(* IEC 61131-3 sources: OLIA-RU/Lirics/OpenPLC_Runtime/Projects/ModbusTCP_slave_test/build, 2 files *)

(* ---- plc.st ---- *)
TYPE
  LOGLEVEL : (CRITICAL, WARNING, INFO, DEBUG) := INFO;
END_TYPE

FUNCTION_BLOCK LOGGER
  VAR_INPUT
    TRIG : BOOL;
    MSG : STRING;
    LEVEL : LOGLEVEL := INFO;
  END_VAR
  VAR
    TRIG0 : BOOL;
  END_VAR

  IF TRIG AND NOT TRIG0 THEN
  {{
   LogMessage(GetFbVar(LEVEL),(char*)GetFbVar(MSG, .body),GetFbVar(MSG, .len));
  }}
  END_IF;
  TRIG0:=TRIG;
END_FUNCTION_BLOCK

FUNCTION_BLOCK python_eval
  VAR_INPUT
    TRIG : BOOL;
    CODE : STRING;
  END_VAR
  VAR_OUTPUT
    ACK : BOOL;
    RESULT : STRING;
  END_VAR
  VAR
    STATE : DWORD;
    BUFFER : STRING;
    PREBUFFER : STRING;
    TRIGM1 : BOOL;
    TRIGGED : BOOL;
  END_VAR

  {extern void __PythonEvalFB(int, PYTHON_EVAL*);__PythonEvalFB(0, data__);}
END_FUNCTION_BLOCK

FUNCTION_BLOCK python_poll
  VAR_INPUT
    TRIG : BOOL;
    CODE : STRING;
  END_VAR
  VAR_OUTPUT
    ACK : BOOL;
    RESULT : STRING;
  END_VAR
  VAR
    STATE : DWORD;
    BUFFER : STRING;
    PREBUFFER : STRING;
    TRIGM1 : BOOL;
    TRIGGED : BOOL;
  END_VAR

  {extern void __PythonEvalFB(int, PYTHON_EVAL*);__PythonEvalFB(1,(PYTHON_EVAL*)(void*)data__);}
END_FUNCTION_BLOCK

FUNCTION_BLOCK python_gear
  VAR_INPUT
    N : UINT;
    TRIG : BOOL;
    CODE : STRING;
  END_VAR
  VAR_OUTPUT
    ACK : BOOL;
    RESULT : STRING;
  END_VAR
  VAR
    py_eval : python_eval;
    COUNTER : UINT;
    _TMP_ADD10_OUT : UINT;
    _TMP_EQ13_OUT : BOOL;
    _TMP_SEL15_OUT : UINT;
    _TMP_AND7_OUT : BOOL;
  END_VAR

  _TMP_ADD10_OUT := ADD(COUNTER, 1);
  _TMP_EQ13_OUT := EQ(N, _TMP_ADD10_OUT);
  _TMP_SEL15_OUT := SEL(_TMP_EQ13_OUT, _TMP_ADD10_OUT, 0);
  COUNTER := _TMP_SEL15_OUT;
  _TMP_AND7_OUT := AND(_TMP_EQ13_OUT, TRIG);
  py_eval(TRIG := _TMP_AND7_OUT, CODE := CODE);
  ACK := py_eval.ACK;
  RESULT := py_eval.RESULT;
END_FUNCTION_BLOCK

PROGRAM OLIA_examle
  VAR
    TestVar AT %QW0 : INT := 0;
  END_VAR
  VAR
    CTU0 : CTU;
    TON0 : TON;
    TP0 : TP;
    _TMP_XOR20_OUT : BOOL;
    R_TRIG1 : R_TRIG;
  END_VAR

  _TMP_XOR20_OUT := XOR(TON0.Q, True);
  TP0(IN := _TMP_XOR20_OUT, PT := T#1000ms);
  TON0(IN := TP0.Q, PT := T#500ms);
  R_TRIG1(CLK := TON0.Q);
  CTU0(CU := R_TRIG1.Q, R := CTU0.Q, PV := 100);
  TestVar := CTU0.CV;
END_PROGRAM

CONFIGURATION Config0

  RESOURCE Res0 ON PLC
    TASK task0(INTERVAL := T#20ms,PRIORITY := 0);
    PROGRAM instance0 WITH task0 : OLIA_examle;
  END_RESOURCE
END_CONFIGURATION

(* ---- generated_plc.st ---- *)
PROGRAM OLIA_examle
  VAR
    TestVar AT %QW0 : INT := 0;
  END_VAR
  VAR
    CTU0 : CTU;
    TON0 : TON;
    TP0 : TP;
    _TMP_XOR20_OUT : BOOL;
    R_TRIG1 : R_TRIG;
  END_VAR

  _TMP_XOR20_OUT := XOR(TON0.Q, True);
  TP0(IN := _TMP_XOR20_OUT, PT := T#1000ms);
  TON0(IN := TP0.Q, PT := T#500ms);
  R_TRIG1(CLK := TON0.Q);
  CTU0(CU := R_TRIG1.Q, R := CTU0.Q, PV := 100);
  TestVar := CTU0.CV;
END_PROGRAM

CONFIGURATION Config0

  RESOURCE Res0 ON PLC
    TASK task0(INTERVAL := T#20ms,PRIORITY := 0);
    PROGRAM instance0 WITH task0 : OLIA_examle;
  END_RESOURCE
END_CONFIGURATION
